// TwinCAT 3 PLC project TestJig
// ProgramVersion: 3.1.4023.0
// libraries:
//   Tc2_Standard, * (Beckhoff Automation GmbH)
//   Tc2_System, * (Beckhoff Automation GmbH)
//   Tc3_Module, * (Beckhoff Automation GmbH)
//   VisuDialogs, * (System)
//   VisuSymbols,3.5.10.0,System
// project tree:
//   DUTs/ sEncoder.TcDUT
//   / GlobalTextList.TcGTLO, ImagePool.TcIPO (not stored), I_O_Idle_Task.TcTTO (not stored), PlcTask.TcTTO, VisualizationManager.TcVMO (not stored), VISU_TASK.TcTTO
//   GVLs/ HMI_IO.TcGVL, Motor_IO.TcGVL, Module_IO.TcGVL, TS.TcGVL
//   POUs/ Laser.TcPOU, MAIN.TcPOU, Encoder.TcPOU, MC.TcPOU, Safety.TcPOU
//   VISUs/ V_AI.TcVIS, V_DI.TcVIS, V_DO.TcVIS, V_Encoder.TcVIS, V_Main.TcVIS, V_MainScreen.TcVIS, V_MC.TcVIS, VPP.TcVIS, V_Safety.TcVIS
// real-time tasks:
//   TASK PlcTask: cycle T#10ms, priority 20, ADS port 350
//   TASK VISU_TASK: cycle T#200000us, priority 30, ADS port 351
//   TASK PLC communication Task: cycle T#10ms, priority 60, ADS port 352
// I/O:
//   DEVICE Device 1 (EtherCAT), AmsNetId 192.168.1.123.2.1
//     Term 8 (EK1100) [EK1100 EtherCAT Coupler (2A E-Bus)]
//       Term 10 (EL6900) [EL6900, TwinSAFE PLC]
//       Term 12 (EL1904) [EL1904, 4 Ch. Safety Input 24V, TwinSAFE]
//         modules: Module 1 (FSOES)
//       Term 13 (EL2904) [EL2904, 4 Ch. Safety Output 24V, 0.5A, TwinSAFE]
//         modules: Module 1 (FSOES), Module 2 (DO)
//       Term 14 (EL1004) [EL1004 4Ch. Dig. Input 24V, 3ms]
//       Term 15 (EL1008) [EL1008 8Ch. Dig. Input 24V, 3ms]
//       Term 16 (EL2004) [EL2004 4Ch. Dig. Output 24V, 0.5A]
//       Term 17 (EL5001) [EL5001 1Ch. SSI Encoder]
//       Term 18 (EL3152) [EL3152 2Ch. Ana Input 4-20mA]
//       Term 18 (EL9011) [EL9011 End Terminal]
//   DEVICE Device 2 (EtherCAT Automation Protocol), AmsNetId 192.168.1.123.3.1
//     Box 7 (Publisher)
// variable links:
//   Device 1 (EtherCAT) <-> Device 1 (EtherCAT)/Term 8 (EK1100)/Term 10 (EL6900)
//     Term 8 (EK1100)/Term 12 (EL1904)/Module 1 (FSOES)/RxPDO/FSOE <-> ConnectionInputs/Message_50 TxPDO
//   Device 1 (EtherCAT) <-> Device 1 (EtherCAT)/Term 8 (EK1100)/Term 12 (EL1904)
//     Term 8 (EK1100)/Term 10 (EL6900)/ConnectionOutputs/Message_50 RxPDO <-> Module 1 (FSOES)/TxPDO/FSOE
//   Device 1 (EtherCAT) <-> Device 1 (EtherCAT)/Term 8 (EK1100)/Term 13 (EL2904)
//     Term 8 (EK1100)/Term 10 (EL6900)/ConnectionInputs/Message_77 TxPDO <-> Module 1 (FSOES)/RxPDO/FSOE
//     Term 8 (EK1100)/Term 10 (EL6900)/ConnectionOutputs/Message_77 RxPDO <-> Module 1 (FSOES)/TxPDO/FSOE
//   TestJig/TestJig Instance <-> Device 1 (EtherCAT)/Term 8 (EK1100)/Term 18 (EL3152)
//     PlcTask Inputs/Laser.nLaserRawValue <-> AI Standard Channel 1/Value
//     PlcTask Inputs/Laser.sLaserError <-> AI Standard Channel 1/Status/Error

CONFIGURATION TestJig
    RESOURCE PLC ON TwinCAT3
        TASK PlcTask(INTERVAL := T#10ms, PRIORITY := 20);
        TASK VISU_TASK(INTERVAL := T#200000us, PRIORITY := 30);
        PROGRAM MAIN WITH PlcTask : MAIN;
        PROGRAM VisuElems_Visu_Prg WITH VISU_TASK : VisuElems.Visu_Prg;
    END_RESOURCE
END_CONFIGURATION

// ---- DUTs/sEncoder.TcDUT
TYPE sEncoder :
STRUCT
	bDataError  	AT %I* : BIT;
	bFrameError 	AT %I* : BIT;
	bPowerFail		AT %I* : BIT;
	bSyncError		AT %I* : BIT;
	bPDOState		AT %I* : BIT;
	bPDOToggle		AT %I* : BIT;
	uCounter		AT %I* : UDINT;
	bInputToggle	AT %I* : BIT;
END_STRUCT
END_TYPE

// ---- GVLs/HMI_IO.TcGVL
{attribute 'qualified_only'}
VAR_GLOBAL
	//MC Lamps
	bMCStartLamp	: BOOL;
	bMCStopLamp		: BOOL;
	bMCResetEstop	: BOOL; 
	bMCForwardlamp	: BOOL;
	bMCReserveLamp	: BOOL;
	
	//Safety Lamp
	bSafetyResetLamp	: BOOL;
	
	//DO Lamps
	bDOStartLamp	: BOOL;
	bDOForwardLamp	: BOOL;
	bDOResetLamp	: BOOL;
	bDOReverselamp	: BOOL;
	
	iEncoderOffset  : REAL;
	

END_VAR

// ---- GVLs/Motor_IO.TcGVL
{attribute 'qualified_only'}
VAR_GLOBAL
	
END_VAR

// ---- GVLs/Module_IO.TcGVL
{attribute 'qualified_only'}
VAR_GLOBAL
	iResetButton		AT %I* 	: BOOL;	//Reset Button EL1008 I1
	iBypassSwitch		AT %I* 	: BOOL; //Bypass Switch EL1008 I2
	iTestInput			AT %I* 	: ARRAY[3..6] OF BOOL; //EL1008 I3- I6 FOR testing sensors
	iMotorOverLoad		AT %I* 	: BOOL; //EL1008 I7
	iMotorContactorAux	AT %I* 	: BOOL; //EL1008 I8
	
	oStartLamp			AT %Q* 	: BOOL; //Start button Lamp EL2004 I1
	oForward			AT %Q* 	: BOOL; //Selector switch EL2004 I2
	oResetButton		AT %Q* 	: BOOL; //Reset button Lamp EL2004 I3
	oReverse			AT %Q* 	: BOOL; //Selector switch EL2004 I4
	
	iStartButton		AT %I* 	: BOOL;	//Start Button EL1004 I1
	iStopButton			AT %I* 	: BOOL;	//Stop Button EL1004 I2
	iForward			AT %I* 	: BOOL;	//Selector Switch Forward EL1004 I3
	iReverse			AT %I* 	: BOOL;	//Selector Switch Reverse EL1004 I4
	
	nLaserValue			AT %I*  : REAL;
	nEncoderValue		AT %I*  : UDINT;
END_VAR

// ---- GVLs/TS.TcGVL
{attribute 'qualified_only'}
VAR_GLOBAL
	//Safety Mat
	iSafetyMat1		AT %I* : BOOL; //Safety Mat input 1 
	iSafetyMat2		AT %I* : BOOL; //Safety Mat input 2 
	iSafetyMatAlarm AT %I* : BOOL; // For E-stop or Safety mat alarm
	
	// E-Stop
	iEStop1 		AT %I* : BOOL; // E-Stop Contact 1
	iEStop2 		AT %I* : BOOL; // E-Stop Contact 2
	iEStopAlarm 	AT %I* : BOOL; 
	
	//From Std module Reset.sds
	oReset			AT %Q* : BOOL;
	
	//Run and Err Ack sds
	oRunInput		AT %Q* : BOOL;
	oRunOutput		AT %Q* : BOOL;
	oErrAckInput	AT %Q* : BOOL;
	oErrAckOutput	AT %Q* : BOOL;
	
	// For Motor control MotorOn.sds
	oMotorON		AT %Q* : BOOL;
	iMotorEStop 	AT %I* : BOOL;
	iMotorOkToRun 	AT %I* : BOOL;
	iForward		AT %I* : BOOL;
	iReverse		AT %I* : BOOL;
	oForward		AT %Q* : BOOL;
	oReverse		AT %Q* : BOOL;
	oOverload		AT %Q* : BOOL;
	oContactor		AT %Q* : BOOL;

END_VAR

// ---- POUs/MAIN.TcPOU
PROGRAM MAIN
VAR
	tonFlash : TON;
	tDelay	: TIME := T#500MS;
END_VAR

//Opening other POUs
Encoder();
Safety();
Laser();
MC();

//LED Flash control
tonFlash(IN:=NOT tonFlash.Q, PT:=tDelay, Q=>);

END_PROGRAM

// ---- POUs/Encoder.TcPOU
PROGRAM Encoder
VAR
	//Encoder1 : Link to EL5001
	nRawData 		: REAL;
	nScaling 		: REAL;
	nOffset 		: REAL;
	nVoltage 		: REAL;
	testEncoder		: sEncoder;
	sScalingTable 	: ARRAY[0..2] OF WSTRING := ["Stacker Table WAN", "WT3 WAN"];
	iScaleTable		: INT := 0;
END_VAR



IF iScaleTable=0 THEN
	nScaling := 0.0004224;
ELSIF  iScaleTable=1 THEN
	nScaling := 0.0002636080;
ELSE
	nScaling := 0.0004224;
END_IF
 
//nCounter := UDINT_TO_REAL(Encoder1.
//testEncoder.bInputToggle := TRUE;
nVoltage := UDINT_TO_REAL(testEncoder.uCounter) * nScaling + nOffset;
	
(*
IF Module_IO.iBypassSwitch THEN
	testEncoder.bInputToggle := TRUE;
	nVoltage := UDINT_TO_REAL(testEncoder.uCounter) * nScaling;
ELSE
	testEncoder.bInputToggle := FALSE;
END_IF
*)

END_PROGRAM

// ---- POUs/Safety.TcPOU
PROGRAM Safety
VAR
	rTrig : R_Trig;
	tonDelay : TON;
END_VAR


IF TS.iSafetyMat1 AND TS.iSafetyMat2 AND TS.iEStop1 AND TS.iEStop2 THEN
	TS.iSafetyMatAlarm := FALSE;
ELSE
	TS.iSafetyMatAlarm := TRUE;
END_IF



IF NOT TS.iEStop1 OR NOT TS.iEStop2 OR MC.iState = 100 THEN
	TS.oReset := FALSE;
	TS.oErrAckInput := FALSE;
	TS.oErrAckOutput := FALSE;
	TS.oRunInput := FALSE;
	TS.oRunOutput := FALSE;
	//Module_IO.iRelaySwitch := FALSE;
ELSIF Module_IO.iResetButton THEN // Reset button, toggle only
	TS.oErrAckInput := TRUE;
	TS.oErrAckOutput := TRUE;
	//Module_IO.iRelaySwitch := TRUE;
	TS.oRunInput := TRUE;
	TS.oRunOutput := TRUE;
END_IF



(********* Bypass to be used for screens  **********
IF HMI_IO.iDigital[1] THEN //Bypass/Run switch
	TS.oRunInput := TRUE;
	TS.oRunOutput := TRUE;
	HMI_IO.iMotorControl[5] := TRUE;
ELSE
	TS.oRunInput := FALSE;
	TS.oRunOutput := FALSE;
	HMI_IO.iMotorControl[5] := FALSE;
END_IF
    **********************************************)

END_PROGRAM

// ---- POUs/MC.TcPOU
PROGRAM MC
VAR
	bMotorControlEnabled 	: BOOL := FALSE;
	iState					: INT := 0;
	sState					: WSTRING;
	tonAuxON				: TON;
	bEstopEngaged			: BOOL;
	tonDelay				: TON;
	tDelay					: TIME := T#5S;
	sAlarm					: WSTRING := " ";
	tReversing				: TIME;
	tForward				: TIME;
	bTimerOff				: BOOL := FALSE;
END_VAR

Inputs();

CASE iState OF
	0: sState := "E-Stop engaged";
			//HMI_IO.bDOStartLamp := FALSE;
			Module_IO.oStartLamp := FALSE;
			TS.oMotorON := FALSE;
			TS.oReverse := FALSE;
			TS.oForward := FALSE;
			tonDelay(IN:=FALSE);
	  	IF NOT bEstopEngaged THEN 
			sState := "E-Stop disengaged";
			IF Module_IO.iResetButton THEN 
				TS.oReset := TRUE;
				iState := 5;
	  		END_IF
		ELSE
			sState := "E-Stop engaged";
		END_IF
		IF Main.tonFlash.Q THEN
			//HMI_IO.bMCResetEstop := NOT HMI_IO.bMCResetEstop;
			Module_IO.oResetButton := NOT Module_IO.oResetButton;
		END_IF
		bTimerOff := FALSE;
	
	5:	sState := "Ready to Start Motor";
		TS.oReset := FALSE;
		bTimerOff := FALSE;
	    IF bMotorControlEnabled AND NOT bEstopEngaged THEN 
			tonDelay(IN:=FALSE);
			TS.oReverse := FALSE;
			TS.oForward := FALSE;
			//HMI_IO.bMCResetEstop := FALSE;
			Module_IO.oResetButton := FALSE;
			TS.oMotorON := FALSE;
			
			IF Main.tonFlash.Q THEN
				//HMI_IO.bDOStartLamp := NOT HMI_IO.bDOStartLamp;
				Module_IO.oStartLamp := NOT Module_IO.oStartLamp;
			END_IF
			IF Module_IO.iStartButton THEN
				iState := 10;
			END_IF
		ELSIF bEstopEngaged THEN
			iState := 0;
		END_IF
		
	10: sState := "Motor Forward/Reverse Control Enabled";
		TS.oMotorON := TRUE;
		Module_IO.oStartLamp := TRUE;
		tonDelay(IN:=FALSE);
		bTimerOff := FALSE;
		IF bMotorControlEnabled AND NOT bEstopEngaged THEN
			IF Module_IO.iForward THEN 
				iState := 20;
			ELSIF Module_IO.iReverse THEN
				iState := 30;
			END_IF
		ELSIF bEstopEngaged THEN
			iState := 0;
		ELSIF NOT bMotorControlEnabled THEN
			iState := 5;
		END_IF
		
	
	20: sState := "Running Forward";
		
		IF TS.oForward AND bMotorControlEnabled THEN
			bTimerOff := TRUE;
			tonDelay(IN:=Module_IO.iForward, PT:=tDelay, Q=>, ET=>tForward); //Safety when swtching the motor to reverse
			IF tonDelay.Q THEN 
				Module_IO.oForward := TRUE;
				//tonDelay(IN:=FALSE);
				bTimerOff := FALSE;
				(* tonAuxOn(IN:=TRUE, PT:=T#20S, Q=>, ET=>);
				IF Module_IO.iMotorContactorAux AND NOT tonAuxOn.Q THEN 
					tonAuxON(IN:=FALSE);
				ELSE
					sAlarm := "Forward Control issue, Press Emergency Stop";
					Module_IO.oForward := FALSE;
					iState := 100;
				END_IF  *)
			END_IF
		ELSE 
			Module_IO.oForward := FALSE;
			tonDelay(IN:=FALSE);
			iState := 10;
		END_IF
		IF NOT bMotorControlEnabled THEN
			iState := 5;
		ELSIF bEstopEngaged THEN
			iState := 0;
		END_IF
		
	30: sState := "Running Reverse";
	
		IF TS.oReverse AND bMotorControlEnabled THEN
			bTimerOff := TRUE;
			tonDelay(IN:=Module_IO.iReverse, PT:=tDelay, Q=>, ET=>tReversing); //Safety when swtching the motor to reverse
			IF tonDelay.Q THEN 
				Module_IO.oReverse := TRUE;
				//tonDelay(IN:=FALSE);
				bTimerOff := FALSE;
				(*tonAuxOn(IN:=TRUE, PT:=T#20S, Q=>, ET=>);
				IF Module_IO.iMotorContactorAux AND NOT tonAuxOn.Q THEN 
					tonAuxON(IN:=FALSE);
				ELSE
					sAlarm := "Reverser Control issue, Press Emergency Stop";
					Module_IO.oForward := FALSE;
					iState := 100;
				END_IF *)
			END_IF
		ELSE 
			Module_IO.oReverse := FALSE;
			tonDelay(IN:=FALSE);
			iState := 10;
		END_IF
		IF NOT bMotorControlEnabled THEN
			iState := 5;
		ELSIF bEstopEngaged THEN
			iState := 0;
		END_IF
		
    100: 
		sState := "Alarm: {sALARM}";
		TS.oMotorON := FALSE;
		bTimerOff := FALSE;
		Module_IO.oStartLamp := FALSE;
		IF Main.tonFlash.Q THEN
			//HMI_IO.bMCResetEstop := NOT HMI_IO.bMCResetEstop;
			Module_IO.oResetButton := NOT Module_IO.oResetButton;
		END_IF
	
END_CASE

//First thing to check in case motor is not running
bMotorControlEnabled := Module_IO.iStopButton;// AND NOT Module_IO.iMotorOverLoad;
bEstopEngaged := NOT TS.iEStop1 OR NOT TS.iEStop2;
TS.oOverload := FALSE; //Indicator Only

ACTION Inputs:
//From Twinsafe

TS.oForward := Module_IO.iForward;
TS.oReverse := Module_IO.iReverse;

Module_IO.oForward := TS.iForward;
Module_IO.oReverse := TS.iReverse;

//TS.oContactor := Module_IO.iMotorContactorAux;
TS.oOverload := Module_IO.iMotorOverLoad;
END_ACTION

END_PROGRAM

// ---- POUs/Laser.TcPOU
PROGRAM Laser
VAR
	nLaserRawValue 	AT %I* 	: INT := 0;
	nLaserOffset			: INT := 200;
	tmpVal					: INT;
	sLaserError		AT %I*	: BOOL;
END_VAR


IF nLaserRawValue > 16#6C00 THEN
	Module_IO.nLaserValue:= 0;
ELSE
	tmpVal:= (WORD_TO_INT(nLaserRawValue * 4800 / 16#6C00)+ nLaserOffset);
	Module_IO.nLaserValue:= tmpVal;
END_IF

END_PROGRAM

// ---- GlobalTextList.TcGTLO
TEXTLIST GlobalTextList
  183 = '%d'
  353 = '%f'
  4 = '%s'
  275 = '<'
  313 = '>'
  571 = 'AI'
  436 = 'Alarm'
  206 = 'Authorised Personnel Use Only'
  918 = 'before terminating any input'
  356 = 'Black'
  776 = 'Bypass'
  547 = 'Bypass NIU'
  869 = 'Close'
  954 = 'CURRENTVISU'
  957 = 'DI'
  536 = 'DO'
  207 = 'DO NOT STARE INTO BEAM'
  678 = 'E-Stop'
  952 = 'E-Stop 1'
  677 = 'E-Stop 2'
  470 = 'EK1100'
  620 = 'EK1904'
  256 = 'EL1004'
  376 = 'EL1008'
  521 = 'EL6900'
  343 = 'Encoder'
  272 = 'Encoder Reading'
  194 = 'E_Stop 1'
  703 = 'F0'
  978 = 'F1'
  891 = 'F2'
  290 = 'F3'
  968 = 'F4'
  587 = 'F5'
  411 = 'F6'
  997 = 'Forward'
  30 = 'Forward NIU'
  953 = 'Input I1'
  820 = 'Input I2'
  689 = 'Input I3'
  416 = 'Input I3+'
  919 = 'Input I3-'
  305 = 'Input I4'
  111 = 'Input I4+'
  763 = 'Input I4-'
  70 = 'Input I5'
  158 = 'Input I6'
  590 = 'Input I7'
  825 = 'Input I8'
  636 = 'Issue:'
  564 = "Issue: PC Isn't reading/connecting to EK1100. Used a new one but same result."
  157 = 'Issue: We cannot connect to EK1100. Used a new one but same result.'
  518 = 'Laser Distance (mm)'
  494 = 'LASER LIGHT'
  860 = 'Laser Light '
  357 = 'Laser Light Donot Stare into Beam'
  836 = 'Main'
  359 = 'MC'
  72 = 'Navigate through pages/screens'
  310 = 'Offset'
  517 = 'or output in any module'
  235 = 'Output O1'
  910 = 'Output O2'
  749 = 'Output O3'
  669 = 'Output O4'
  34 = 'Output O5'
  327 = 'Output O6'
  164 = 'Output O7'
  250 = 'Output O8'
  743 = 'Overload'
  841 = 'Raw'
  955 = 'Raw Value'
  516 = 'Reset'
  574 = 'Reset E-Stop'
  984 = 'Reset NIU'
  524 = 'Reverse'
  652 = 'Reverse NIU'
  395 = 'Run TS'
  826 = 'Safety'
  31 = 'Scale'
  960 = 'Scaleing'
  348 = 'Scaling'
  489 = 'Start'
  830 = 'Start/Running'
  388 = 'Stop'
  301 = 'Switch OFF power supply to PLC'
  839 = 'Test'
  449 = 'Test Button 1'
  882 = 'Time ON delay %s'
  926 = 'TS Channel'
  637 = 'TS Channel 3'
  398 = 'TS Channel 4'
  770 = 'using buttons'
  977 = 'WAN Scale:'
  365 = 'WAN Scale: 0.0002636080'
  228 = 'We need ideas to program in this test jig.'
  220 = 'We now have connections to I/Os, We need ideas to program in this test jig.'
  970 = 'White'
END_TEXTLIST

// ---- VISUs/V_AI.TcVIS
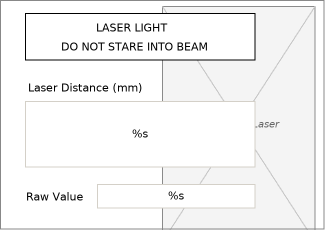
VISUALIZATION V_AI  // 325x230
    Image (162,6 153x236), image: ImagePool.Laser
    Rectangle (25,13 230x47)
    Label (93,20 183x21), "LASER LIGHT"
    Label (58,39 183x21), "DO NOT STARE INTO BEAM"
    Label (25,73 167x30), "Laser Distance (mm)"
    Textfield (25,101 230x66), "%s", text variable: Module_IO.nLaserValue
    Label (23,182 71x30), "Raw Value"
    Textfield (97,184 158x24), "%s", text variable: Laser.nLaserRawValue
END_VISUALIZATION

// ---- VISUs/V_DI.TcVIS
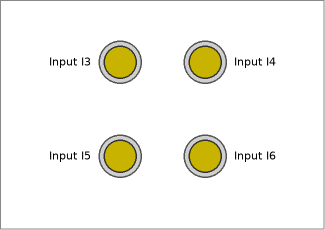
VISUALIZATION V_DI  // 325x230
    Lamp1 (95,37 50x50), variable: Module_IO.iTestInput[3], style: Lamp-Lamp1-Yellow
    Lamp1 (180,37 50x50), variable: Module_IO.iTestInput[4], style: Lamp-Lamp1-Yellow
    Lamp1 (95,131 50x50), variable: Module_IO.iTestInput[5], style: Lamp-Lamp1-Yellow
    Lamp1 (180,131 50x50), variable: Module_IO.iTestInput[6], style: Lamp-Lamp1-Yellow
    Label (40,47 60x30), "Input I3"
    Label (40,141 60x30), "Input I5"
    Label (225,47 60x30), "Input I4"
    Label (225,141 60x30), "Input I6"
END_VISUALIZATION

// ---- VISUs/V_DO.TcVIS
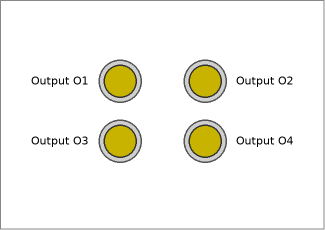
VISUALIZATION V_DO  // 325x230
    Lamp1 (95,56 50x50), variable: HMI_IO.bDOStartLamp, style: Lamp-Lamp1-Yellow
    Lamp1 (180,56 50x50), variable: HMI_IO.bMCForwardlamp, style: Lamp-Lamp1-Yellow
    Lamp1 (95,116 50x50), variable: HMI_IO.bDOResetLamp, style: Lamp-Lamp1-Yellow
    Lamp1 (180,116 50x50), variable: HMI_IO.bDOReverselamp, style: Lamp-Lamp1-Yellow
    Label (25,66 70x30), "Output O1"
    Label (25,126 70x30), "Output O3"
    Label (230,66 70x30), "Output O2"
    Label (230,126 70x30), "Output O4"
END_VISUALIZATION

// ---- VISUs/V_Encoder.TcVIS
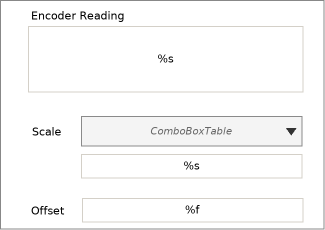
VISUALIZATION V_Encoder  // 325x230
    Textfield (28,26 275x66), "%s", text variable: Encoder.nVoltage
        p4168582468: Encoder.nVoltage
    Label (28,1 118x30), "Encoder Reading"
    Label (29,117 52x30), "Scale"
    Textfield (81,154 221x24), "%s", text variable: Encoder.nScaling
        p4168582468: Encoder.nScaling
    Label (28,196 52x30), "Offset"
    Textfield (82,198 221x24), "%f", text variable: Encoder.nOffset
        OnMouseClick: write Encoder.nOffset via VisuDialogs.Numpad, min 1, max 5000, title "Encoder Offset"
    ComboBoxTable (81,116 221x30), variable: Encoder.iScaleTable, data array: Encoder.sScalingTable
        p3854506369: Encoder.sScalingTable[INDEX]
END_VISUALIZATION

// ---- VISUs/V_Main.TcVIS
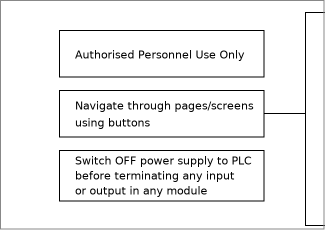
VISUALIZATION V_Main  // 325x230
    Rectangle (59,150 205x51)
    Rectangle (59,90 205x47)
    Rectangle (59,30 205x47)
    Label (72,98 185x21), "Navigate through pages/screens"
    Label (72,153 191x31), "Switch OFF power supply to PLC"
    Label (72,168 181x31), "before terminating any input"
    Label (72,47 183x21), "Authorised Personnel Use Only"
    Line (305,12) (305,225)
    Line (264,113) (305,113)
    Line (305,12) (325,12)
    Line (305,225) (325,225)
    Label (72,115 177x21), "using buttons"
    Label (72,183 146x20), "or output in any module"
END_VISUALIZATION

// ---- VISUs/V_MainScreen.TcVIS
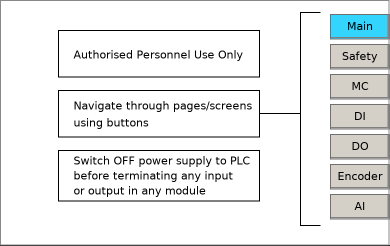
VISUALIZATION V_MainScreen  // 390x246
    Button (330,14 60x25), "Main"
        OnMouseClick: FrameSelectionChange Selection=SelectedFrame=ca35193f-53d6-45b7-b8b5-0860b53cf110, GlobSel=AssignType=Directly, SelType=Locally
    Button (330,44 60x25), "Safety"
        OnMouseClick: FrameSelectionChange Selection=SelectedFrame=ca35193f-53d6-45b7-b8b5-0860b53cf110, Selection=1, GlobSel=AssignType=Directly, SelType=Locally
    Button (330,74 60x25), "MC"
        OnMouseClick: FrameSelectionChange Selection=SelectedFrame=ca35193f-53d6-45b7-b8b5-0860b53cf110, Selection=2, GlobSel=AssignType=Directly, SelType=Locally
    Button (330,104 60x25), "DI"
        OnMouseClick: FrameSelectionChange Selection=SelectedFrame=ca35193f-53d6-45b7-b8b5-0860b53cf110, Selection=3, GlobSel=AssignType=Directly, SelType=Locally
    Button (330,134 60x25), "DO"
        OnMouseClick: FrameSelectionChange Selection=SelectedFrame=ca35193f-53d6-45b7-b8b5-0860b53cf110, Selection=4, GlobSel=AssignType=Directly, SelType=Locally
    Button (330,164 60x25), "Encoder"
        OnMouseClick: FrameSelectionChange Selection=SelectedFrame=ca35193f-53d6-45b7-b8b5-0860b53cf110, Selection=5, GlobSel=AssignType=Directly, SelType=Locally
    Button (330,194 60x25), "AI"
        OnMouseClick: FrameSelectionChange Selection=SelectedFrame=ca35193f-53d6-45b7-b8b5-0860b53cf110, Selection=6, GlobSel=AssignType=Directly, SelType=Locally
    Line (0,245) (390,245)
    Frame (0,0 320x230)
        shows V_Main()
        shows V_Safety()
        shows V_MC()
        shows V_DI()
        shows V_DO()
        shows V_Encoder()
        shows V_AI()
END_VISUALIZATION

// ---- VISUs/V_MC.TcVIS
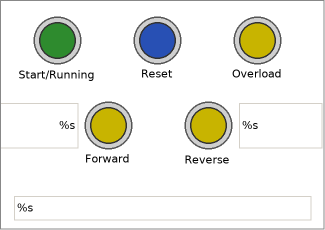
VISUALIZATION V_MC  // 325x230
    Lamp1 (30,13 55x55), variable: Module_IO.oStartLamp, style: Lamp-Lamp1-Green
    Label (9,60 95x30), "Start/Running"
    Lamp1 (130,13 55x55), variable: Module_IO.oResetButton, style: Lamp-Lamp1-Blue
    Label (108,59 98x30), "Reset"
    Lamp1 (81,98 55x55), variable: Module_IO.oForward, style: Lamp-Lamp1-Yellow
    Lamp1 (181,98 55x55), variable: Module_IO.oReverse, style: Lamp-Lamp1-Yellow
    Label (64,144 87x30), "Forward"
    Label (166,145 82x30), "Reverse"
    Textfield (14,196 297x24), "%s", text variable: MC.sState
    Textfield (0,103 78x45), "%s", text variable: MC.tForward, invisible if: NOT (Module_IO.iForward AND MC.bTimerOff)
    Textfield (239,103 83x45), "%s", text variable: MC.tReversing, invisible if: NOT (Module_IO.iReverse AND MC.bTimerOff)
    Lamp1 (230,13 55x55), variable: Module_IO.iMotorOverLoad, style: Lamp-Lamp1-Yellow
    Label (208,59 98x30), "Overload"
END_VISUALIZATION

// ---- VISUs/VPP.TcVIS
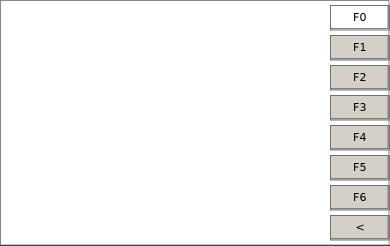
VISUALIZATION VPP  // 390x246
    Button (330,5 60x25), "F0"
    Button (330,35 60x25), "F1"
    Button (330,65 60x25), "F2"
    Button (330,95 60x25), "F3"
    Button (330,125 60x25), "F4"
    Button (330,155 60x25), "F5"
    Button (330,185 60x25), "F6"
    Line (0,245) (390,245)
    Button (330,215 60x25), "<"
        OnMouseClick: change screen: V_Safety
END_VISUALIZATION

// ---- VISUs/V_Safety.TcVIS
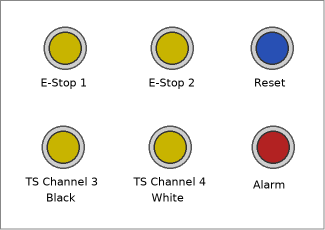
VISUALIZATION V_Safety  // 325x230
    Lamp1 (38,122 50x50), variable: TS.iSafetyMat1, style: Lamp-Lamp1-Yellow
    Lamp1 (145,122 50x50), variable: TS.iSafetyMat2, style: Lamp-Lamp1-Yellow
    Label (15,167 94x30), "TS Channel 3"
    Label (21,121 70x30)
    Label (26,183 70x30), "Black"
    Lamp1 (248,122 50x50), variable: TS.iSafetyMatAlarm, style: Lamp-Lamp1-Red
    Label (234,170 70x30), "Alarm"
    Label (123,167 94x30), "TS Channel 4"
    Label (133,183 70x30), "White"
    Lamp1 (40,23 50x50), variable: TS.iEStop1, style: Lamp-Lamp1-Yellow
    Lamp1 (147,23 50x50), variable: TS.iEStop2, style: Lamp-Lamp1-Yellow
    Label (17,68 94x30), "E-Stop 1"
    Label (125,68 94x30), "E-Stop 2"
    Lamp1 (247,23 50x50), variable: Module_IO.oResetButton, style: Lamp-Lamp1-Blue
    Label (235,68 70x30), "Reset"
END_VISUALIZATION
